{attribute 'linkalways'} 
{attribute 'no_explicit_call' := 'This FB is a CLASS and must be accessed using methods or properties'}
{attribute 'enable_dynamic_creation'}
FUNCTION_BLOCK Parameter EXTENDS Disposable IMPLEMENTS I_Parameter
VAR
	_name : T_MAXSTRING;
	_data : I_Datatype;
	_parent : I_HostParameters;
	_connectedTo : I_LinkSource;
	eventEmitter : EventEmitter;
	metadataHost : MetadataHost(THIS^, eventEmitter);
END_VAR

METHOD PUBLIC Accept
VAR_INPUT
	Visitor : I_ParameterVisitor;
END_VAR
Visitor.VisitParameter(THIS^);
END_METHOD

METHOD PUBLIC AddMetadata : I_HostMetadata
VAR_INPUT
	Name : T_MAXSTRING;
	Data : I_Datatype;
END_VAR
Metadatum.AddDataAsMetadata(Name, Data);
AddMetadata := THIS^;
END_METHOD

PROPERTY PUBLIC Connected : BOOL
GET
Connected := _connectedTo <> 0;
END_GET
END_PROPERTY

PROPERTY PUBLIC Data : I_Datatype
GET
Data := _data;
END_GET
END_PROPERTY

METHOD PUBLIC Disconnect
IF NOT Connected THEN
	RETURN;
END_IF

_connectedTo := 0;
_data.ClearReference();
END_METHOD

METHOD FB_init : BOOL
VAR_INPUT
	bInitRetains : BOOL; // if TRUE, the retain variables are initialized (warm start / cold start)
	bInCopyCode : BOOL;  // if TRUE, the instance afterwards gets moved into the copy code (online change)
	Name : T_MAXSTRING;
	Data : I_Datatype;
	Parent : I_HostParameters;
END_VAR
_name := Name;
_data := Data;
RegisterWithParent(Parent);
END_METHOD

PROPERTY PUBLIC Metadatum : I_Metadatum
GET
Metadatum := metadataHost;
END_GET
END_PROPERTY

PROPERTY PUBLIC Name : T_MAXSTRING
GET
Name := _name;
END_GET
END_PROPERTY

METHOD PUBLIC OffEvent
VAR_INPUT
	EventName : T_MaxString;
	EventHandler : I_EventHandler;
END_VAR
eventEmitter.OffEvent(EventName, EventHandler);
END_METHOD

METHOD PUBLIC OnceEvent
VAR_INPUT
	EventName : T_MaxString;
	EventHandler : I_EventHandler;
END_VAR
eventEmitter.OnceEvent(EventName, EventHandler);
END_METHOD

METHOD PUBLIC OnEvent
VAR_INPUT
	EventName : T_MaxString;
	EventHandler : I_EventHandler;
END_VAR
eventEmitter.OnEvent(EventName, EventHandler);
END_METHOD

PROPERTY PUBLIC Parent : I_HostParameters
GET
Parent := _parent;
END_GET
END_PROPERTY

METHOD PUBLIC RegisterWithParent
VAR_INPUT
	Parent : I_HostParameters;
END_VAR
IF Parent = 0 THEN
	RETURN;
END_IF

THIS^._parent := Parent;
Parent.Parameters.AddParameter(THIS^);
END_METHOD

METHOD PUBLIC SerializeWith
VAR_INPUT
	Serializer : I_Serializer;
END_VAR
Serializer.StartObject();
Serializer.AddKeyString('name', _name);
Serializer.Addkey('datatype');
_data.SerializeTypeWith(Serializer);
Serializer.AddkeyObject('value', _data);
metadataHost.SerializeWith(Serializer);
Serializer.EndObject();
END_METHOD

METHOD PUBLIC TryConnectTo : BOOL
VAR_INPUT
	Source : I_LinkSource;
END_VAR
IF NOT _data.TryMakeReferenceTo(Source.Data) THEN
	RETURN;
END_IF

_connectedTo := Source;
TryConnectTo := TRUE;
END_METHOD

METHOD PUBLIC TryDeserializeFrom : BOOL
VAR_INPUT
	Deserializer : I_Deserializer;
	Feedback : I_DeserializerFeedback;
END_VAR
VAR
	parameterDeserializer : I_Deserializer;
END_VAR
IF Connected THEN 
	RETURN; // the parameter is acting as a port, so it should not apply any deserialized data
END_IF

TryDeserializeFrom := _data.TryDeserializeFrom(Deserializer, Feedback);
END_METHOD

END_FUNCTION_BLOCK

(* stored: Version 1.1.0.1, ProductVersion 3.1.4024.13
   POU Parameter: Id {bad9d0de-f058-492f-999d-54e5404f5ee7}, SpecialFunc None
   Folder Constructor: Id {0fb344eb-1953-45be-b6c3-92152d218a7e}
   Method Accept: Id {04a7a62c-6cae-4a7b-a4b3-bef44a984181}
   Method AddMetadata: Id {25053516-d7c2-0af4-0961-423bd581adcd}
   Property Connected: Id {a0c5d22a-7a99-0a95-05c0-bcc57086a9a5}
   Get Get: Id {d9838e1e-e20e-0710-06ad-8a8390a58b30}
   Property Data: Id {1f0486d5-d52a-49ba-a054-faae67bb8741}
   Get Get: Id {118654b5-095d-4f42-9385-6c7e9f708a99}
   Method Disconnect: Id {7cf594b9-9c1b-0381-1f1d-904078f3abf4}
   Method FB_init: Id {da38514d-cea0-4e20-8400-9e2e3dc6adf5}
   Property Metadatum: Id {0afbb18b-4575-4881-a00d-2f3c3483d254}
   Get Get: Id {748178ca-1637-419f-898e-77a3e58ebcf6}
   Property Name: Id {fe024c09-ed38-43b7-9187-f3c7a41f5351}
   Get Get: Id {323b22ce-44b5-400d-92c1-461c45c75128}
   Method OffEvent: Id {2b223bcc-14e5-4367-98d3-d5ec05befd3c}
   Method OnceEvent: Id {6cc392a4-a097-4bcb-96ae-4087b3a20dec}
   Method OnEvent: Id {1c00bb5e-1161-4d75-8ee0-6ac931b47410}
   Property Parent: Id {9a294379-51fa-4591-9330-fbd292b4b9e4}
   Get Get: Id {8535d94d-ca38-4631-9748-58404968af33}
   Method RegisterWithParent: Id {e6732e8a-d3e0-45aa-991b-c9093e562e20}
   Method SerializeWith: Id {e13da5d9-f146-4f8c-80ad-7d2fd4163be7}
   Method TryConnectTo: Id {743a3410-1b48-0def-15ce-d2570b172de0}
   Method TryDeserializeFrom: Id {038b54a1-ee3e-487e-a187-8053c58b8e83} *)
